// Mitsubishi GX Works2 project: Test   PLC: Q03UDV

// task Task_01 (event TRUE, interval 0, priority 31): POU_01

PROGRAM POU_01
VAR
  STATE : INT;
END_VAR
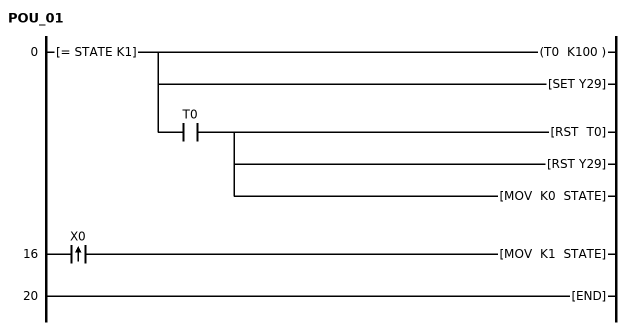
0     LD=     STATE K1
      OUT     T0 K100
      SET     Y29
      AND     T0
      RST     T0
      RST     Y29
      MOV     K0 STATE
16    LDP     X0
      MOV     K1 STATE
20    END
END_PROGRAM
